ABB RAPID module: Calib_Def_wobj_kiste_1.modx

MODULE Calib_Def_wobj_kiste_1(READONLY)
 LOCAL CONST string dataName := "wobj_kiste_1";
 LOCAL CONST string mechUnitRef := "ROB_1";
 LOCAL CONST string toolRef := "tool_calib";
 LOCAL CONST robtarget pWobj_U_PointX1 := [[505.5807,-235.7003,187.013],[3.416703E-06,0.01712747,-0.9998533,4.872382E-06],[-1,-1,-1,0],[8.999999E+09,8.999999E+09,8.999999E+09,8.999999E+09,8.999999E+09,8.999999E+09]];
 LOCAL CONST robtarget pWobj_U_PointX2 := [[504.4584,46.79197,185.8413],[2.468211E-05,0.01713352,-0.9998532,3.899744E-07],[0,0,0,0],[8.999999E+09,8.999999E+09,8.999999E+09,8.999999E+09,8.999999E+09,8.999999E+09]];
 LOCAL CONST robtarget pWobj_U_PointY1 := [[250.3679,-237.6252,184.7016],[4.869041E-05,0.01713056,-0.9998533,3.487103E-06],[-1,-1,-1,0],[8.999999E+09,8.999999E+09,8.999999E+09,8.999999E+09,8.999999E+09,8.999999E+09]];
 !------------------------------------------------------------------------------
 !<auto-generated>
 !This code was generated by a tool.

 !<auto-generated>
 !Changes to this file may cause incorrect behavior and will be lost if
 !the code is regenerated.
 !</auto-generated>
 !------------------------------------------------------------------------------



 ! 31 Jan 2022 10:40:53 by admin from ABB Robotics FlexPendant
 ! Old Value: [FALSE,TRUE,"",[[0,0,0],[1,0,0,0]],[[0,0,0],[1,0,0,0]]]
 !


ENDMODULE
